// TIA Portal V20 export
// export: Created 2025-12-01T14:57:17.3804296Z, ExportSetting None, DisplayName Totally Integrated Automation Portal, DisplayVersion V20 Update 3, DisplayName TIA Portal Openness, DisplayVersion V20 Update 3, DisplayName TIA Portal Version Control Interface, DisplayVersion V20 Update 3, DisplayName STEP 7 Professional, DisplayVersion V20 Update 3, DisplayName STEP 7 Safety, DisplayVersion V20 Update 2, DisplayName WinCC Basic/Comfort/Advanced, DisplayVersion V20 Update 3, DisplayName WinCC Professional, DisplayVersion V20 Update 3, DisplayName WinCC Unified, DisplayVersion V20 Update 3
DATA_BLOCK "DB936_Datos_VAR_DANFOSS_PN"   // DB936
{ S7_Optimized_Access := 'FALSE' }
// stored: AutoNumber false
   VAR RETAIN
      Danfoss : Array[0..255] of Struct
         STW_Danfoss { S7_SetPoint := 'True'} : "Danfoss_STW_PN";
         Actual_Speed : Int;
         Dig_Input { S7_SetPoint := 'True'} : "Danfoss_Dig_Input_PN";
         ACC : Int;   // 50->0,5sg; 100->1sg; 500->5sg; 1000->10sg
         DCC : Int;   // 50->0,5sg; 100->1sg; 500->5sg; 1000->10sg
      END_STRUCT;
   END_VAR
BEGIN
   Danfoss[0..255].ACC := 50;
   Danfoss[0..255].DCC := 50;
END_DATA_BLOCK
